FUNCTION_BLOCK PUBLIC FB_PizzaItalianStyle IMPLEMENTS I_Pizza
VAR_INPUT
END_VAR
VAR_OUTPUT
END_VAR
VAR
END_VAR

METHOD GetDescription : STRING
GetDescription := 'Pizza Italian Style:';
END_METHOD

METHOD GetPrice : LREAL
GetPrice := 4.5;
END_METHOD

END_FUNCTION_BLOCK

(* stored: Version 1.1.0.1, ProductVersion 3.1.4022.16
   POU FB_PizzaItalianStyle: Id {544fb8f7-abc4-48db-b83e-66402b2145dc}, SpecialFunc None
   Method GetDescription: Id {9c935248-32b0-46aa-bb8d-93068080127c}
   Method GetPrice: Id {6f8072c3-e000-430d-9e6f-606d9a40c2d7} *)
